(* IEC 61131-3 sources: Word/plc-course/09-math-and-data-handling/labs/starter, 3 files *)

(* ---- 09-1-scaling-function.st ---- *)
(* Lab 09-1: A general scaling function, F_Scale.
   Module 09 (Maths, comparison, data movement and bit manipulation).
   STARTER - the function's inputs and the program's interface are declared
   for you; write the logic where it says TODO, then run:
     python3 tools/plctest.py 09-math-and-data-handling/labs/starter/09-1-scaling-function.st

   Raw-count convention (as in Module 14): 0..27648 = 4..20 mA. *)

FUNCTION F_Scale : REAL
  VAR_INPUT
    In     : REAL;   (* the value to convert *)
    InMin  : REAL;   (* input value that corresponds to OutMin *)
    InMax  : REAL;   (* input value that corresponds to OutMax *)
    OutMin : REAL;   (* result when In = InMin *)
    OutMax : REAL;   (* result when In = InMax *)
    Clamp  : BOOL;   (* TRUE: keep the result inside the output range *)
  END_VAR
  (* TODO: add a VAR ... END_VAR block for any local variables you need. *)

  (* TODO: straight-line scaling with divide-by-zero protection and an
     optional clamp. OutMin may be larger than OutMax.
     Replace this placeholder line with your logic. *)
  F_Scale := 0.0;
END_FUNCTION

PROGRAM ScalingDemo
  VAR (* I/O *)
    LevelRaw AT %IW0 : INT;   (* LT-101 tank level, raw counts from the analog input card *)
    SpeedAO  AT %QW0 : INT;   (* SC-103 drive speed reference, raw counts: 0..27648 = 4..20 mA *)
    ValveAO  AT %QW1 : INT;   (* FV-102 valve demand, raw counts: 0 = 4 mA = fully OPEN *)
  END_VAR
  VAR (* settings: configuration of the card, the transmitter and the drive *)
    RawAt4mA   : REAL := 0.0;      (* raw count the card gives at 4 mA *)
    RawAt20mA  : REAL := 27648.0;  (* raw count the card gives at 20 mA *)
    DriveMinHz : REAL := 0.0;      (* drive speed at 4 mA (drive parameter) *)
    DriveMaxHz : REAL := 50.0;     (* drive speed at 20 mA (drive parameter) *)
  END_VAR
  VAR (* HMI values *)
    Level_m      : REAL;           (* LT-101 level in metres, NOT clamped *)
    LevelPct     : REAL;           (* LT-101 level in % of range, clamped 0..100 for the bar graph *)
    SpeedRef_Hz  : REAL;           (* speed setpoint entered on the HMI *)
    ValveCmd_Pct : REAL;           (* valve opening demand: 0 = closed, 100 = fully open *)
  END_VAR
  VAR CONSTANT
    LEVEL_MIN_M : REAL := 0.5;     (* LT-101 range: 0.5 m at 4 mA (the tapping is 0.5 m above the floor) ... *)
    LEVEL_MAX_M : REAL := 4.5;     (* ... 4.5 m at 20 mA *)
    AO_RAW_4MA  : REAL := 0.0;     (* analog output raw count for 4 mA *)
    AO_RAW_20MA : REAL := 27648.0; (* analog output raw count for 20 mA *)
  END_VAR

  (* TODO: calculate the four values with F_Scale (see the lab requirements
     in the Module 09 README). Replace these placeholder lines. *)
  Level_m := 0.0;
  LevelPct := 0.0;
  SpeedAO := 0;
  ValveAO := 0;
END_PROGRAM

CONFIGURATION Config0
  RESOURCE Res0 ON PLC
    TASK MainTask(INTERVAL := T#10ms, PRIORITY := 0);
    PROGRAM Inst0 WITH MainTask : ScalingDemo;
  END_RESOURCE
END_CONFIGURATION

(* ---- 09-2-reject-tracking.st ---- *)
(* Lab 09-2: Conveyor reject tracking with a bit shift register.
   Module 09 (Maths, comparison, data movement and bit manipulation).
   STARTER - the interface is declared for you; write the logic where it
   says TODO, then run:
     python3 tools/plctest.py 09-math-and-data-handling/labs/starter/09-2-reject-tracking.st

   Each bit of TrackWord stands for one position on the belt:

      bit:      15  ...  6   5   4   3   2   1   0
      position: 15  ...  6   5   4   3   2   1   0 (camera)
                              ^ reject gate (RejectPos = 5)

   MATIEC has no bit access such as TrackWord.5: use masks and shifts,
   for example (TrackWord AND SHL(WORD#16#0001, n)) <> 0 to test bit n. *)

PROGRAM RejectTracking
  VAR (* I/O *)
    EncoderPulse AT %IX0.0 : BOOL;  (* one pulse per pitch, from a prox on the drive sprocket *)
    InspectFail  AT %IX0.1 : BOOL;  (* camera at position 0: TRUE = the part in front of it failed *)
    ResetPB      AT %IX0.2 : BOOL;  (* clear the tracking after the belt has been emptied by hand *)
    RejectGate   AT %QX0.0 : BOOL;  (* reject pusher at position RejectPos *)
  END_VAR
  VAR (* settings and HMI values *)
    RejectPos   : INT := 5;         (* pitches from the camera to the reject gate, 1..15 *)
    TrackWord   : WORD;             (* bit n TRUE = the part n pitches past the camera is bad *)
    RejectCount : DINT;             (* bad parts that have reached the reject gate *)
  END_VAR
  VAR (* suggested internal variables: add, rename or remove as you like *)
    PulseEdge : R_TRIG;             (* the belt has moved one pitch *)
  END_VAR

  (* TODO: mark, shift, test the gate bit, count and reset (see the lab
     requirements in the Module 09 README). Replace these placeholder lines. *)
  PulseEdge(CLK := EncoderPulse);
  TrackWord := WORD#16#0000;
  RejectGate := FALSE;
  RejectCount := 0;
END_PROGRAM

CONFIGURATION Config0
  RESOURCE Res0 ON PLC
    TASK MainTask(INTERVAL := T#10ms, PRIORITY := 0);
    PROGRAM Inst0 WITH MainTask : RejectTracking;
  END_RESOURCE
END_CONFIGURATION

(* ---- 09-3-flow-totaliser.st ---- *)
(* Lab 09-3: Flow totaliser.
   Module 09 (Maths, comparison, data movement and bit manipulation).
   STARTER - the interface is declared for you; add your own internal
   variables and write the logic where it says TODO, then run:
     python3 tools/plctest.py 09-math-and-data-handling/labs/starter/09-3-flow-totaliser.st

   Every scan:  increment [m3] = flow [m3/h] x scan time [h]

   MATIEC notes: TIME_TO_REAL and TIME_TO_LREAL return SECONDS here (CODESYS
   returns milliseconds), so a ratio such as
   TIME_TO_LREAL(TaskCycle) / TIME_TO_LREAL(T#1h) is the portable way to get
   hours. Conversions between REAL and LREAL are explicit: REAL_TO_LREAL,
   LREAL_TO_REAL, DINT_TO_LREAL, DINT_TO_REAL. TRUNC(x) cuts off the fraction. *)

PROGRAM FlowTotaliser
  VAR (* I/O *)
    ResetPB  AT %IX0.0 : BOOL;       (* reset the totaliser to zero (NO key switch) *)
    PresetPB AT %IX0.1 : BOOL;       (* load PresetValue_m3 into the totaliser (NO) *)
  END_VAR
  VAR (* process value and settings *)
    FlowRate       : REAL;           (* FT-201 flow in m3/h, already scaled (Module 14) *)
    PresetValue_m3 : DINT;           (* whole m3 to load, e.g. the reading of the meter being replaced *)
    TaskCycle      : TIME := T#10ms; (* the task interval: must match the TASK INTERVAL below *)
  END_VAR
  VAR RETAIN (* on a real PLC the totals must survive a power cut *)
    Total_m3     : LREAL;            (* the accurate total, m3 *)
    TotalReal_m3 : REAL;             (* the naive REAL total, m3: for comparison only *)
  END_VAR
  VAR (* outputs for SCADA and the HMI *)
    TotalWhole_m3 : DINT;            (* whole cubic metres of Total_m3, like a meter's counter *)
  END_VAR
  (* TODO: add a VAR ... END_VAR block here for your helper variables
     (MATIEC does not accept an empty VAR block, so none is given). *)

  (* TODO: integrate FlowRate into Total_m3 (accurately) and into
     TotalReal_m3 (the naive REAL way), with reset and preset; then
     TotalWhole_m3. Replace these placeholder lines with your logic. *)
  Total_m3 := 0.0;
  TotalReal_m3 := 0.0;
  TotalWhole_m3 := 0;
END_PROGRAM

CONFIGURATION Config0
  RESOURCE Res0 ON PLC
    TASK MainTask(INTERVAL := T#10ms, PRIORITY := 0);
    PROGRAM Inst0 WITH MainTask : FlowTotaliser;
  END_RESOURCE
END_CONFIGURATION
